// TIA Portal V20 export
TYPE "LER_typeCommunicationInterfaceData"
// stored: Access Published
   STRUCT
      HeartBeat : Byte;
      "Bool" : Array[0..95] of Bool;
      LReal : Array[0..19] of LReal;
   END_STRUCT;
END_TYPE
